# EPICS IOC start-up script: require/3.1.2/siteMods/recsync/1.3.0-9705e52/recsync.iocsh
#- ####################################################
#- ###               RECSYNC    iocsh               ###
#- ####################################################
#- >> Mandatory
#- IOCNAME            - IOCNAME (A-A:B-B)
#- >> Optional
#- TIMEOUT    - RECCAST timeout, Default : 5.0
#- MAXHOLDOFF - RECCAST MaxHoldoff, Default : 5.0
#-
#-
var(reccastTimeout, "$(TIMEOUT=5.0)")
var(reccastMaxHoldoff, "$(MAXHOLDOFF=5.0)")
#-
dbLoadRecords("reccaster.db", "P=$(IOCNAME)-RecSync:")
#-
